// TIA Portal V20 export
FUNCTION "LAH100" : Void   // FC8, FBD
{ S7_Optimized_Access := 'TRUE' }
// stored: SetENOAutomatically false
BEGIN

REGION Network 1: Channel input
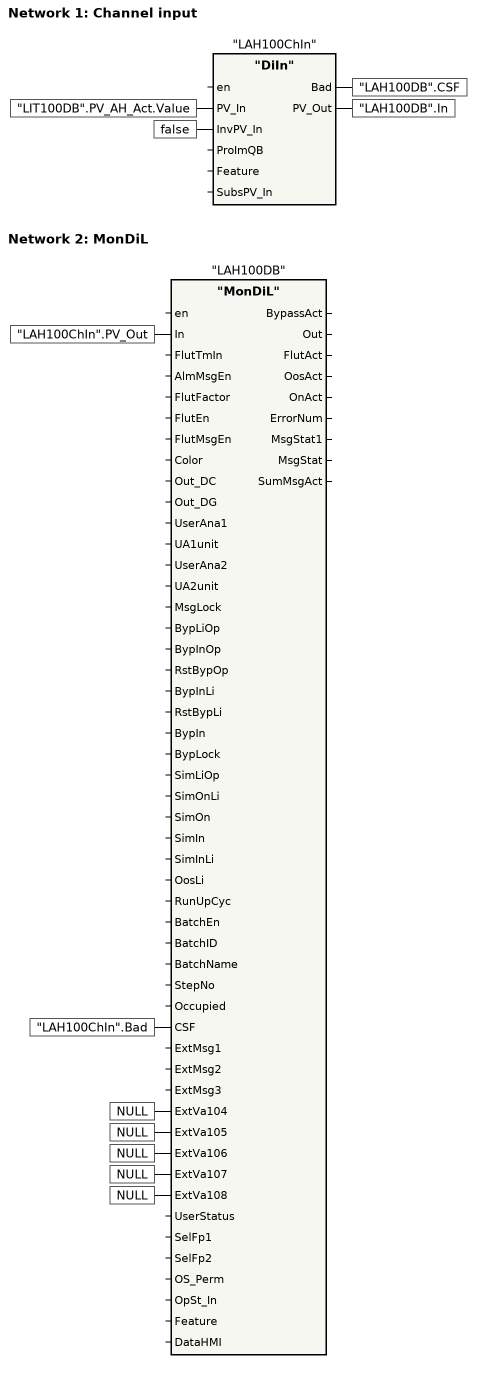
   "LAH100ChIn"(PV_In := "LIT100DB".PV_AH_Act.Value,   // "DiIn"
                InvPV_In := false,
                Bad => "LAH100DB".CSF,
                PV_Out => "LAH100DB".In);
END_REGION

REGION Network 2: MonDiL
   "LAH100DB"(In := "LAH100ChIn".PV_Out,   // "MonDiL"
              CSF := "LAH100ChIn".Bad,
              ExtVa104 := NULL,
              ExtVa105 := NULL,
              ExtVa106 := NULL,
              ExtVa107 := NULL,
              ExtVa108 := NULL);
END_REGION

REGION Network 3: MTP
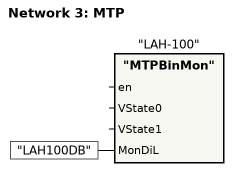
   "LAH-100"(MonDiL := "LAH100DB");   // "MTPBinMon"
END_REGION
END_FUNCTION
